PROGRAM p03_SR1
VAR
	// Set
	S0: BOOL;
	// Reset
	S1: BOOL;
	// Q
	L0: BOOL;
END_VAR

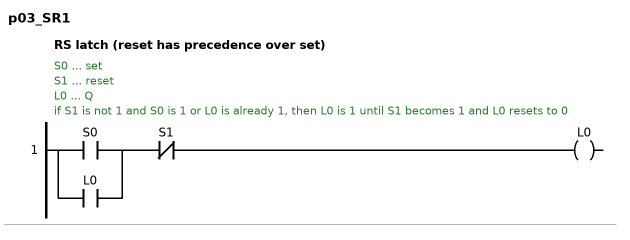
// NETWORK 1: RS latch (reset has precedence over set)
// S0 ... set
// S1 ... reset
// L0 ... Q
// if S1 is not 1 and S0 is 1 or L0 is already 1, then L0 is 1 until S1 becomes 1 and L0 resets to 0
L0 := (S0 OR L0) AND NOT S1;

END_PROGRAM

(* stored: Version 1.1.0.1, ProductVersion 3.1.4024.13
   POU p03_SR1: Id {fea03186-e556-4205-b9dd-38b8e1bc8a99}, SpecialFunc None *)
